// TwinCAT 3 PLC project RedLine
// ProgramVersion: 3.1.4023.0
// libraries:
//   Tc2_Standard, * (Beckhoff Automation GmbH)
//   Tc2_System, * (Beckhoff Automation GmbH)
//   Tc3_Module, * (Beckhoff Automation GmbH)
// project tree:
//   GVLs/ GVL.TcGVL
//   / PlcTask.TcTTO
//   POUs/ MAIN.TcPOU
// real-time tasks:
//   TASK PlcTask: cycle T#10ms, priority 20, ADS port 350
//   TASK PlcTask1: cycle T#10ms, priority 21, ADS port 351

CONFIGURATION RedLine
    RESOURCE PLC ON TwinCAT3
        TASK PlcTask(INTERVAL := T#10ms, PRIORITY := 20);
        PROGRAM MAIN WITH PlcTask : MAIN;
    END_RESOURCE
END_CONFIGURATION

// ---- GVLs/GVL.TcGVL
{attribute 'qualified_only'}
VAR_GLOBAL

//Block States IO
mInSwitch : ARRAY[0..40] OF DINT;
mOutSwitch : ARRAY[0..40] OF DINT;
mInOccupancies : ARRAY[0..40] OF DINT;
mOutOccupancies : ARRAY[0..40] OF DINT;
mInSpeeds : ARRAY[0..40] OF DINT;
mOutSpeeds : ARRAY[0..40] OF DINT;
mInAuthorities : ARRAY[0..40] OF DINT;
mOutAuthorities : ARRAY[0..40] OF DINT;
mInCrossings : ARRAY[0..40] OF DINT;
mOutCrossings : ARRAY[0..40] OF DINT;
mInLeftLights : ARRAY[0..40] OF DINT;
mOutLeftLights : ARRAY[0..40] OF DINT;
mInRightLights : ARRAY[0..40] OF DINT;
mOutRightLights : ARRAY[0..40] OF DINT;
mInMaintenance : ARRAY[0..40] OF DINT;
mOutMaintenance : ARRAY[0..40] OF DINT;
mInRoute : ARRAY[0..76] OF DINT;
mOutRoute : ARRAY[0..76] OF DINT;
mSpeedLimits : ARRAY[0..44] OF DINT := [70,70,70,70,70,70,70,70,70,70,70,70,70,70,70,70,60,60,55,55,55,55,55,55,55,55,55,55,55,55,55,55,55,55,55,55,55,55,55,70];

END_VAR

// ---- POUs/MAIN.TcPOU
PROGRAM MAIN
VAR

inc1 : DINT := 0;
	
END_VAR

FOR inc1 := 0 TO 40 DO
	//Sets Red Lights
	IF GVL.mInOccupancies[inc1] = 0
	THEN
		GVL.mOutLeftLights[inc1] := 0;
		GVL.mOutRightLights[inc1] := 0;
	//Sets green lights
	ELSE
		GVL.mOutLeftLights[inc1] := 2;
		GVL.mOutRightLights[inc1] := 2;
	END_IF
END_FOR

FOR inc1 := 1 TO 39 DO
	//Sets Yellow Lights
	IF GVL.mInOccupancies[inc1-1] = 0 AND GVL.mInOccupancies[inc1] <> 0
	THEN
		GVL.mOutRightLights[inc1] := 1;
	END_IF
	IF GVL.mInOccupancies[inc1+1] = 0 AND GVL.mInOccupancies[inc1] <> 0
	THEN
	GVL.mOutLeftLights[inc1] := 1;
	END_IF
END_FOR

//0 to 40 correspond to blocks 33 to 71
//copies inputs to outputs for blocks 33 to 71
FOR inc1 := 0 TO 40 DO

	GVL.mOutOccupancies[inc1] := GVL.mInOccupancies[inc1];
	IF GVL.mInSpeeds[inc1] < GVL.mSpeedLimits[inc1]
	THEN
		GVL.mOutSpeeds[inc1] := GVL.mInSpeeds[inc1];
	ELSE
		GVL.mOutSpeeds[inc1] := GVL.mSpeedLimits[inc1];
	END_IF
	GVL.mOutAuthorities[inc1] := GVL.mInAuthorities[inc1];
	GVL.mOutMaintenance[inc1] := GVL.mInMaintenance[inc1];
	GVL.mOutRoute[inc1] := 1;
	
END_FOR

//This copies route over from input to output
FOR inc1 := 0 TO 76 DO

	GVL.mOutRoute[inc1] := GVL.mInRoute[inc1];
	
END_FOR

inc1 := 0;

//This starts the main track logic section

//Crossing Logic
IF GVL.mInOccupancies[14] = 0 THEN
	GVL.mOutCrossings[14] := 1;
ELSE
	GVL.mOutCrossings[14] := 0;
END_IF

//Switch Logic

//Sets switch on block 40
IF GVL.mInMaintenance[5] = 1 
THEN
   IF GVL.mInSwitch[5] = 1
	THEN
		IF GVL.mOutSwitch[5] = 40
		THEN
			GVL.mOutSwitch[5] := 70;
		ELSE
			GVL.mOutSwitch[5] := 40;
		END_IF
		GVL.mInSwitch[5] := 0;
	END_IF
ELSE
    IF GVL.mInOccupancies[6] = 0 THEN
    FOR inc1 := 0 TO 5 DO 
        IF GVL.mInOccupancies[inc1] = 0 THEN
            GVL.mOutSwitch[5] := 40;
            Exit;
        ELSE 
            GVL.mOutSwitch[5] := 70;
        END_IF
    END_FOR
	END_IF
END_IF

//Set switch on block 44
IF GVL.mInMaintenance[10] = 1 
THEN
    IF GVL.mInSwitch[10] = 1
	THEN
		IF GVL.mOutSwitch[10] = 40
		THEN
			GVL.mOutSwitch[10] := 70;
		ELSE
			GVL.mOutSwitch[10] := 40;
		END_IF
		GVL.mInSwitch[10] := 0;
	END_IF
ELSE
    IF GVL.mInOccupancies[9] = 0 THEN
    FOR inc1 := 10 TO 18 DO 
        IF GVL.mInOccupancies[inc1] = 0 THEN
            GVL.mOutSwitch[10] := 66;
            Exit;
        ELSE 
            GVL.mOutSwitch[10] := 42;
        END_IF
    END_FOR
	END_IF
END_IF

//Set switch on block 52
IF GVL.mInMaintenance[18] = 1 
THEN
    IF GVL.mInSwitch[18] = 1
	THEN
		IF GVL.mOutSwitch[18] = 52
		THEN
			GVL.mOutSwitch[18] := 65;
		ELSE
			GVL.mOutSwitch[18] := 52;
		END_IF
		GVL.mInSwitch[18] := 0;
	END_IF
ELSE
    IF GVL.mInOccupancies[32] = 0 THEN
    FOR inc1 := 10 TO 18 DO 
        IF GVL.mInOccupancies[inc1] = 0 THEN
            GVL.mOutSwitch[18] := 52;
            Exit;
        ELSE 
            GVL.mOutSwitch[18] := 65;
        END_IF
    END_FOR
	END_IF
END_IF

END_PROGRAM
